TYPE ST_SubSystemRegistryConv :
(**************************************************************************************
 * 	Application		:	BoxControl Framework
 *	Revision		:	$Revision: 404529 $
 *	Revision date	:	$Date: 2018-04-23 08:21:38 +0200 (Mo., 23 Apr 2018) $
 *	Last changed by	:	$Author: b7bolm $
 *	URL				:	$URL: http://almscdc.swisslog.com/repo/SWPD/Development/BoxControlFramework/20_Release/trunk/01_Software/BCF/BCF/JumpStart/20_Product/10_App/10_Base/10_Lib/10_Conv/01_DUTs/ST_SubSystemRegistryConv.TcDUT $
 *
 *	Purpose			:	Subsystem registration structure.
 *
 * ------------------------------------------------------------------------------------
 *	Copyright Swisslog [IP AG], Switzerland. All rights reserved.
 * 
 * ------------------------------------------------------------------------------------
 *	
 * 	Revision History: 
 *
 * 	VERSION			DATE			INITIALS			DESCRIPTION
 *	0.1				01.01.2001		swl					Example
 *
 **************************************************************************************)
STRUCT
	SubsystemName			: STRING(System.NAME_LENGTH); // Name as string
	rSubsystemData			: REFERENCE TO ST_SubsystemData;
	rSubsystemInterface 	: REFERENCE TO ST_SubsystemInterface;
	rSettingsSubsystem	 	: REFERENCE TO ST_CFG_Subsystem;
	rSubsystem				: REFERENCE TO FB_SubsystemConv;
	HashCode				: UDINT; // HashCode
END_STRUCT
END_TYPE

(* stored: Version 1.1.0.1, ProductVersion 3.1.4022.12
   DUT ST_SubSystemRegistryConv: Id {be9a4680-89b7-41b6-a677-73156d7881b0} *)
